{attribute 'GeneratedUsingTerminal: EP2816-0004-0016'}
{attribute addProperty BoxType "EP2816-0004-0016"}
{attribute addProperty Id "EtcSlaveTerminalBaseDO_Outputs_Channel_1AT %Q*DO_Outputs_Channel_28AC1A9E8DO_Outputs_Channel_2AT %Q*DO_Outputs_Channel_28AC1A9E8WcStateAT %I*WcState_0B2B16F91InfoDataAT %I*InfoData_32EB74EA10"}
{attribute addProperty CRC "3022323835"}
{attribute addProperty Size "27"}
TYPE EP2816_B425007B EXTENDS EtcSlaveTerminalBase :
STRUCT
	{attribute addProperty Name "DO_Outputs_Channel_1"}
	DO_Outputs_Channel_1 : DO_Outputs_Channel_28AC1A9E;
	{attribute addProperty Name "DO_Outputs_Channel_2"}
	DO_Outputs_Channel_2 : DO_Outputs_Channel_28AC1A9E;
	{attribute addProperty Name "WcState"}
	WcState : WcState_0B2B16F9;
	{attribute addProperty Name "InfoData"}
	InfoData : InfoData_32EB74EA;
END_STRUCT
END_TYPE

(* stored: Version 1.2.0.0, ProductVersion 3.1.4024.9
   DUT EP2816_B425007B: Id {d258126f-6fb2-43c4-9996-d50a95aea1b3} *)
